// TIA Portal V17 export
// export: Created 2025-04-11T04:54:24.8026442Z, ExportSetting WithDefaults, DisplayName Totally Integrated Automation Portal, DisplayVersion V17, DisplayName TIA Portal Openness, DisplayVersion V17, DisplayName TIA Portal Version Control Interface, DisplayVersion V17, DisplayName SINAMICS Startdrive Advanced, DisplayVersion V17, DisplayName SINAMICS Startdrive G130, G150, S120, S150, SINAMICS MV, S210, DisplayVersion V17, DisplayName SINAMICS Startdrive G110M, G120, G120C, G120D, G120P, G115D, DisplayVersion V17, DisplayName STEP 7 Professional, DisplayVersion V17, DisplayName STEP 7 Safety, DisplayVersion V17, DisplayName WinCC Advanced, DisplayVersion V17
TYPE "UDT_Ana_Temp"
// stored: IsFailsafeCompliant false
   STRUCT
      IN_SimMode : Bool;   // 模拟模式
      IN_ManualValue : Real;   // 手动设定值
      IN_Enable3Take2 : Bool;   // 启用3取2功能
      OUT_EngValue1 : Real;   // 传感器1工程值
      OUT_EngValue2 : Real;   // 传感器2工程值
      OUT_EngValue3 : Real;   // 传感器3工程值
      OUT_RawCurrent1 : Real;   // 传感器1电流值(mA)
      OUT_RawCurrent2 : Real;   // 传感器2电流值(mA)
      OUT_RawCurrent3 : Real;   // 传感器3电流值(mA)
   END_STRUCT;
END_TYPE
